   _009: NOP   0;

         A     "Temp".If_Up;
         JNB   _006;

         L     "Temp".TriangleUp;
         L     25.0;
         +R;
         T     "Temp".TriangleUp;

   _006: NOP   0;

         L     "Temp".TriangleUp;
         L     999.0;
         >=R;
         JNB   _008;

         T     "Temp".TriangleUp;

         CLR;
         =     "Temp".If_Up;

   _008: NOP   0;

         L     "Temp".TriangleUp;
         L     0.0;
         <=R;
         JNB   _007;

         T     "Temp".TriangleUp;

         SET;
         =     "Temp".If_Up;

   _007: NOP   0;

         L     "Temp".TriangleUp;
         TRUNC;
         T     #For_TriangleUp;

   // квадраты
         L     "Temp".Square;
         L     25.0;
         +R;
         T     "Temp".Square;

         L     999.0;
         >R;
         JNB   _004;

         L     -999.0;
         T     "Temp".Square;

   _004: NOP   0;

         L     -999;
         T     #For_Square;

         L     "Temp".Square;
         L     0;
         >R;
         JNB   _005;

         L     999;
         T     #For_Square;

   _005: NOP   0;

   // Пила
         L     "Temp".Ramp;
         L     20.0;
         +R;
         T     "Temp".Ramp;

         L     "Temp".Ramp;
         L     999.0;
         >R;
         JNB   _003;

         L     -999.0;
         T     "Temp".Ramp;

   _003: NOP   0;

         L     "Temp".Ramp;
         TRUNC;
         T     #For_Ramp;

   // Синуоида
         L     "Temp".Radians;
         L     0.15;
         +R;
         T     "Temp".Radians;
         L     31415.9;
         >R;
         JNB   _002;

         L     "Temp".Radians;
         L     31415.9;
         -R;
         T     "Temp".Radians;

   _002: NOP   0;

   //     ITD
   //      DTR
         L     "Temp".Radians;
         COS;
         L     1000.0;
         *R;
         TRUNC;
         T     #For_SIN;

         L     100.0;
         *R;


   //== Запись в массив оссциллографирования
         CALL  "Wr_OSC"
         ( Var_1  := #For_SIN,
           Var_2  := #For_Ramp,
           Var_3  := #For_Square,
           Var_4  := #For_TriangleUp,
           Var_5  := #CH_05,
           Var_6  := #CH_06,
           Var_7  := #CH_07,
           Var_8  := #CH_08,
           Var_9  := #CH_09,
           Var_10 := #CH_10
         );
END_REGION

REGION Network 2



         A(;
         L     "DB_OSC".Ramp;
         L     1;
         +I;
         T     "DB_OSC".Ramp;
         AN    OV;
         SAVE;
         CLR;
         A     BR;
         );
         A(;
         L     "DB_OSC".Ramp;
         L     5000;
         >I;
         );
         JNB   _001;
         L     0;
         T     "DB_OSC".Ramp;
   _001: NOP   0;
END_REGION
END_FUNCTION

FUNCTION "Wr_OSC" : Void   // FC505, STL
{ S7_Optimized_Access := 'FALSE' }
VERSION : 0.1
// Запись параметров в массив осцилографирования
// Версия 20-10-2014
   VAR_INPUT
      Var_1 : Int;
      Var_2 : Int;
      Var_3 : Int;
      Var_4 : Int;
      Var_5 : Int;
      Var_6 : Int;
      Var_7 : Int;
      Var_8 : Int;
      Var_9 : Int;
      Var_10 : Int;
   END_VAR
   VAR_TEMP
      Tmp_1 : DInt;
      Tmp_2 : DInt;
      Tmp_3 : DInt;
      Tmp_4 : DInt;
      Tmp_5 : DInt;
      Tmp_6 : DInt;
      Tmp_7 : DInt;
      Tmp_Ramp : DInt;
      Ramp : Int;
      Tmp_8 : DInt;
      Tmp_9 : DInt;
      Tmp_10 : DInt;
      RV : Int;
   END_VAR
BEGIN

REGION Network 1
   // 658619651
         A     %DB505.DBX1.0;
         FP    "OSC_Work";
         JNB   STRT;

         CALL  "Ini_Arr"
         ( Reg := 0
         );

   STRT: A     %DB505.DBX1.0;
         JNB   FIN;

   //---------------- Расчёт номера участка
         L     1;
         L     "DB_OSC".Cnt;
         +I;
         T     "DB_OSC".Cnt;
         L     50;
         >I;
         JNB   _NFR;

         L     1;
         T     "DB_OSC".Cnt;

         L     1;
         L     "DB_OSC".Ready;
         +I;
         T     "DB_OSC".Ready;
         L     4;
         >I;
         JNB   _NFR;

         L     1;
         T     "DB_OSC".Ready;

   _NFR: NOP   0;

   //------------------------------------
         L     "DB_OSC".cr_Addr_1;
         T     #Tmp_1;

         L     "DB_OSC".cr_Addr_2;
         T     #Tmp_2;

         L     "DB_OSC".cr_Addr_3;
         T     #Tmp_3;

         L     "DB_OSC".cr_Addr_4;
         T     #Tmp_4;

         L     "DB_OSC".cr_Addr_5;
         T     #Tmp_5;

         L     "DB_OSC".cr_Addr_6;
         T     #Tmp_6;

         L     "DB_OSC".cr_Addr_7;
         T     #Tmp_7;

         L     "DB_OSC".cr_Addr_8;
         T     #Tmp_8;

         L     "DB_OSC".cr_Addr_9;
         T     #Tmp_9;

         L     "DB_OSC".cr_Addr_10;
         T     #Tmp_10;

   //--------------------------------
   // Запись значений в блок данных
   //--------------------------------
         OPN   "DB_OSC";
         L     #Var_1;
         T     DBW [#Tmp_1];
         T     "DB_OSC".Ch_1;

         OPN   "DB_OSC";
         L     #Var_2;
         T     DBW [#Tmp_2];
         T     "DB_OSC".Ch_2;

         OPN   "DB_OSC";
         L     #Var_3;
         T     DBW [#Tmp_3];
         T     "DB_OSC".Ch_3;

         OPN   "DB_OSC";
         L     #Var_4;
         T     DBW [#Tmp_4];
         T     "DB_OSC".Ch_4;

         OPN   "DB_OSC";
         L     #Var_5;
         T     DBW [#Tmp_5];
         T     "DB_OSC".Ch_5;

         OPN   "DB_OSC";
         L     #Var_6;
         T     DBW [#Tmp_6];
         T     "DB_OSC".Ch_6;

         OPN   "DB_OSC";
         L     #Var_7;
         T     DBW [#Tmp_7];
         T     "DB_OSC".Ch_7;

         OPN   "DB_OSC";
         L     #Var_8;
         T     DBW [#Tmp_8];
         T     "DB_OSC".Ch_8;

         OPN   "DB_OSC";
         L     #Var_9;
         T     DBW [#Tmp_9];
         T     "DB_OSC".Ch_9;

         OPN   "DB_OSC";
         L     #Var_10;
         T     DBW [#Tmp_10];
         T     "DB_OSC".Ch_10;

   //------------------------------
   // Пересчёт адресов
   //------------------------------
         L     DINT#16;
         L     "DB_OSC".cr_Addr_1;
         +D;
         T     "DB_OSC".cr_Addr_1;

         L     DINT#16;
         L     "DB_OSC".cr_Addr_2;
         +D;
         T     "DB_OSC".cr_Addr_2;

         L     DINT#16;
         L     "DB_OSC".cr_Addr_3;
         +D;
         T     "DB_OSC".cr_Addr_3;

         L     DINT#16;
         L     "DB_OSC".cr_Addr_4;
         +D;
         T     "DB_OSC".cr_Addr_4;

         L     DINT#16;
         L     "DB_OSC".cr_Addr_5;
         +D;
         T     "DB_OSC".cr_Addr_5;

         L     DINT#16;
         L     "DB_OSC".cr_Addr_6;
         +D;
         T     "DB_OSC".cr_Addr_6;

         L     DINT#16;
         L     "DB_OSC".cr_Addr_7;
         +D;
         T     "DB_OSC".cr_Addr_7;

         L     DINT#16;
         L     "DB_OSC".cr_Addr_8;
         +D;
         T     "DB_OSC".cr_Addr_8;

         L     DINT#16;
         L     "DB_OSC".cr_Addr_9;
         +D;
         T     "DB_OSC".cr_Addr_9;

         L     DINT#16;
         L     "DB_OSC".cr_Addr_10;
         +D;
         T     "DB_OSC".cr_Addr_10;

         L     DINT#16;
         L     "DB_OSC".cr_Addr_Rmp;
         +D;
         T     "DB_OSC".cr_Addr_Rmp;

         L     "DB_OSC".Max_Addr;
         >D;
         JNB   _NAR;

         CALL  "Ini_Arr"
         ( Reg := 1
         );

   _NAR: NOP   0;

   FIN:  NOP   0;
END_REGION
END_FUNCTION

FUNCTION "Ini_Arr" : Void   // FC506, STL
{ S7_Optimized_Access := 'FALSE' }
VERSION : 0.0
// Инициализация параметров осцилографирования
// Версия: 16-10-2014
// Входные параметры:
//   Reg - режим работы программы
//     0 - Задать адреса набора 1 и очистить все массивы
//     1 - Задать адреса набора 1
//     2 - Задать адреса набора 2
   VAR_INPUT
      Reg : Int;
   END_VAR
   VAR_TEMP
      Addr : DInt;
   END_VAR
BEGIN

REGION Network 1: SCL network

   //--------------------------------------
   // Начальные адреса массивов
   //--------------------------------------
         L     DINT#448;
         T     "DB_OSC".cr_Addr_1;
         L     DINT#3648;
         T     "DB_OSC".cr_Addr_2;
         L     DINT#6848;
         T     "DB_OSC".cr_Addr_3;
         L     DINT#10048;
         T     "DB_OSC".cr_Addr_4;
         L     DINT#13248;
         T     "DB_OSC".cr_Addr_5;
         L     DINT#16448;
         T     "DB_OSC".cr_Addr_6;
         L     DINT#19648;
         T     "DB_OSC".cr_Addr_7;
         L     DINT#22848;
         T     "DB_OSC".cr_Addr_8;
         L     DINT#26048;
         T     "DB_OSC".cr_Addr_9;
         L     DINT#29248;
         T     "DB_OSC".cr_Addr_10;
         L     DINT#32448;
         T     "DB_OSC".cr_Addr_Rmp;

         L     DINT#35632;
         T     "DB_OSC".Max_Addr;

   //--------------------------------------
   // Первая инициализация
   //--------------------------------------
         L     #Reg;
         L     0;
         ==I;
         JCN   A7d1;

   //--------------------------------------
   // Очистка массивов
   //--------------------------------------
         L     0;
         T     "DB_OSC".Ready;
         T     "DB_OSC".Cnt;
         T     "DB_OSC".Ramp;

         L     "DB_OSC".cr_Addr_1;
         T     #Addr;

   A7d3: L     #Addr;
         L     "DB_OSC".Max_Addr;
         <=D;
         JCN   A7d1;

         OPN   "DB_OSC";
         L     DINT#0;
         T     DBW [#Addr];

         L     #Addr;
         L     DINT#16;
         +D;
         T     #Addr;
         JU    A7d3;

   A7d1: NOP   0;

         SAVE;
         CLR;
END_REGION
END_FUNCTION

FUNCTION "OSC_BS_GP" : Void   // FC511, STL
{ S7_Optimized_Access := 'FALSE' }
VERSION : 0.1
   VAR_OUTPUT
      Ch_01 : Int;   // Данные для канала 1
      Ch_02 : Int;   // Данные для канала 2
      Ch_03 : Int;   // Данные для канала 3
      Ch_04 : Int;   // Данные для канала 4
      Ch_05 : Int;   // Данные для канала 5
      Ch_06 : Int;   // Данные для канала 6
      Ch_07 : Int;   // Данные для канала 7
      Ch_08 : Int;   // Данные для канала 8
      Ch_09 : Int;   // Данные для канала 9
      Ch_10 : Int;   // Данные для канала 10
   END_VAR
   VAR_TEMP
      Tmp_DI : DInt;
   END_VAR
BEGIN

REGION Network 1

   //======================== #CH_01
         L     "SU".su_Iq_M1H_fs;
         L     10.0;
         *R;
         RND;
         T     #Tmp_DI;
         L     <??.?>;
         T     #Ch_01;

   //======================== #CH_02
         L     "SU".su_W_M1H_fs;
         L     10.0;
         *R;
         RND;
         T     #Tmp_DI;
         L     <??.?>;
         T     #Ch_02;

   //======================== #CH_03
         L     "SU".su_LH;
         L     10.0;
         *R;
         RND;
         T     #Tmp_DI;
         L     <??.?>;
         T     #Ch_03;

   //======================== #CH_04
         L     "SU".su_LC;
         L     10.0;
         *R;
         RND;
         T     #Tmp_DI;
         L     <??.?>;
         T     #Ch_04;

   //======================== #CH_05
         L     "SU".su_W_S_fs;
         L     10.0;
         *R;
         RND;
         T     #Tmp_DI;
         L     <??.?>;
         T     #Ch_05;

   //======================== #CH_06
         L     "SU".su_Job_C;
         L     DINT#10;
         /D;
         T     #Tmp_DI;
         L     <??.?>;
         T     #Ch_06;


   //      L     "SU".su_Iq_S_fs
   //      L     "SU".su_W_C_fs
   ///      L     1.000000e+001
   //      *R
   //      RND
   //      T     #Tmp_DI
   //      L     LW     2

   //======================== #CH_07
         L     "Work".ug_Pov_Tk;
         T     #Ch_07;

   //      L     "SU".su_LH
   //      L     1.000000e+001
   //      *R
   //      RND
   //      T     #Tmp_DI
   //      L     LW     2

   //======================== #CH_08
         L     "Work".Reg_WC;
         L     100;
         *I;
         T     #Ch_08;

         A     "AP".ap_Gudok;
         JNB   _NGD;

         L     -100;
         T     #Ch_08;

   _NGD: NOP   0;

         A     "AP".ap_ODK;
         JNB   _NOD;

         L     700;
         T     #Ch_08;

   _NOD: NOP   0;

   //      L     "SU".su_LC
   //      L     1.000000e+001
   //      *R
   //      RND
   //     T     #Tmp_DI
   //      L     LW     2

   //======================== #CH_09
         L     "BD".Mas_Basket;
         L     10.0;
         *R;
         RND;
         T     #Tmp_DI;
         L     <??.?>;
         T     #Ch_09;

   //======================== #CH_10
   //      L     "SU".su_Iq_S_fs
         L     "Work".ABS_H;
         L     10.0;
         *R;
         RND;
         T     #Tmp_DI;
         L     <??.?>;
         T     #Ch_10;
END_REGION
END_FUNCTION

FUNCTION "FC514" : Void   // FC514, STL
TITLE = Блок сопряжения осц-фа для ОЭ
{ S7_Optimized_Access := 'FALSE' }
VERSION : 0.1
   VAR_OUTPUT
      Ch_01 : Int;   // Данные для канала 1
      Ch_02 : Int;   // Данные для канала 2
      Ch_03 : Int;   // Данные для канала 3
      Ch_04 : Int;   // Данные для канала 4
      Ch_05 : Int;   // Данные для канала 5
      Ch_06 : Int;   // Данные для канала 6
      Ch_07 : Int;   // Данные для канала 7
      Ch_08 : Int;   // Данные для канала 8
      Ch_09 : Int;   // Данные для канала 9
      Ch_10 : Int;   // Данные для канала 10
   END_VAR
   VAR_TEMP
      Tmp_DI : DInt;
   END_VAR
BEGIN

REGION Network 1

   //======================== #CH_01
         L     "SU".su_Iq_M1H_fs;
         L     10.0;
         *R;
         RND;
         T     #Tmp_DI;
         L     <??.?>;
         T     #Ch_01;

   //======================== #CH_02
         L     "SU".su_W_M1H_fs;
         L     10.0;
         *R;
         RND;
         T     #Tmp_DI;
         L     <??.?>;
         T     #Ch_02;

   //======================== #CH_03
         L     "SU".su_Iq_S_fs;
         L     10.0;
         *R;
         RND;
         T     #Tmp_DI;
         L     <??.?>;
         T     #Ch_03;

   //======================== #CH_04
         L     "SU".su_W_S_fs;
         L     10.0;
         *R;
         RND;
         T     #Tmp_DI;
         L     <??.?>;
         T     #Ch_04;

   //======================== #CH_05
         L     "SU".su_Iq_C_fs;
         L     10.0;
         *R;
         RND;
         T     #Tmp_DI;
         L     <??.?>;
         T     #Ch_05;

   //======================== #CH_06
         L     "SU".su_W_C_fs;
         L     10.0;
         *R;
         RND;
         T     #Tmp_DI;
         L     <??.?>;
         T     #Ch_06;

   //======================== #CH_07
         L     "SU".su_LH;
         L     10.0;
         *R;
         RND;
         T     #Tmp_DI;
         L     <??.?>;
         T     #Ch_07;

   //======================== #CH_08
         L     "SU".su_LC;
         L     10.0;
         *R;
         RND;
         T     #Tmp_DI;
         L     <??.?>;
         T     #Ch_08;

   //======================== #CH_09
         L     "SU".su_Iq_C_fs;
         L     10.0;
         *R;
         RND;
         T     #Tmp_DI;
         L     <??.?>;
         T     #Ch_09;

   //======================== #CH_10
         L     "BD".Mas_TS_cr;
         L     10.0;
         *R;
         RND;
         T     #Tmp_DI;
         L     <??.?>;
         T     #Ch_10;
END_REGION
END_FUNCTION

ORGANIZATION_BLOCK "Main"   // OB1, LAD, ProgramCycle
TITLE = "Main Program Sweep (Cycle)"
{ S7_Optimized_Access := 'TRUE' }
VERSION : 0.1
   VAR_INPUT
      Initial_Call : Bool;   // Initial call of this OB
      Remanence : Bool;   // =True, if remanent data are available
   END_VAR
BEGIN
END_ORGANIZATION_BLOCK

ORGANIZATION_BLOCK "Cyclic interrupt"   // OB35, STL, CyclicInterrupt
{ S7_Optimized_Access := 'TRUE' }
VERSION : 0.1
   VAR_INPUT
      Initial_Call : Bool;   // Initial call of this OB
      Event_Count : Int;   // Events discarded
   END_VAR
BEGIN

REGION Network 1
         CALL  "OSC";
END_REGION
END_ORGANIZATION_BLOCK